PROGRAM MAIN
VAR
END_VAR

END_PROGRAM

(* stored: Version 1.1.0.1
   POU MAIN: Id {faf53572-4d15-4b0f-a977-48da430dcc6d} *)
